// TIA Portal project "Proportional Controller for a Water tank" (V16)
// Vorlageprojekt für das Buch mit Zielsystem S7-1200

(* hardware
DEVICE "S7-1200-Station_1"  S7-1200 Station
   slot 0: "Baugruppenträger_0"  Rack  V1.0
   slot 1: "PLC_1"  CPU 1211C DC/DC/DC  6ES7 211-1AE40-0XB0  V4.1
*)

// ===== PLC "PLC_1"  CPU 1211C DC/DC/DC =====

VAR_GLOBAL   // PLC tag table "Standard-Variablentabelle"
   "xPbStart" AT %I0.0 : Bool;
   "xPbReset" AT %I0.1 : Bool;
   "xPbStop" AT %I0.2 : Bool;
   "xPbStartLed" AT %Q0.0 : Bool;
   "xPbResetLed" AT %Q0.1 : Bool;
   "xPbStopLed" AT %Q0.2 : Bool;
   "rSetpoint" AT %ID38 : Real;
   "rSensorWaterLevel" AT %ID30 : Real;
   "diSP" AT %QD38 : DInt;
   "diPV" AT %QD42 : DInt;
   "rValveFill" AT %QD30 : Real;
   "rValveDischarge" AT %QD34 : Real;
   "xStateStart" AT %M0.0 : Bool;
   "rError" AT %MD2 : Real;
   "rErrorABS" AT %MD6 : Real;
   "rKp" AT %MD10 : Real;
   "rSetpoint_Cm" AT %MD30 : Real;
   "rWaterLevel_Cm" AT %MD34 : Real;
   "xSelectorManual" AT %I0.5 : Bool;
   "xSelectorAuto" AT %I0.4 : Bool;
   "xModeManual" AT %M0.1 : Bool;
   "xModeAuto" AT %M0.2 : Bool;
   "xStep10_EnableRegulator" AT %M0.4 : Bool;
   "xStep30_Discharge" AT %M0.6 : Bool;
   "xStep40_End" AT %M0.7 : Bool;
   "xStep20_LevelCheck" AT %M1.0 : Bool;
   "xAlarm" AT %M0.3 : Bool;
   "xFIOReset" AT %I0.3 : Bool;
   "Clock_Byte" AT %MB100 : Byte;
   "Clock_10Hz" AT %M100.0 : Bool;
   "Clock_5Hz" AT %M100.1 : Bool;
   "Clock_2.5Hz" AT %M100.2 : Bool;
   "Clock_2Hz" AT %M100.3 : Bool;
   "Clock_1.25Hz" AT %M100.4 : Bool;
   "Clock_1Hz" AT %M100.5 : Bool;
   "Clock_0.625Hz" AT %M100.6 : Bool;
   "xPulse" AT %M100.7 : Bool;
   "xStep0_Init" AT %M0.5 : Bool;
   "xMem_0" AT %M1.1 : Bool;
   "diLowerLimit" AT %MD18 : DInt;
   "diupperLimit" AT %MD22 : DInt;
END_VAR

DATA_BLOCK "DB_Regulator"   // DB1
{ S7_Optimized_Access := 'TRUE' }
VERSION : 0.1
   VAR RETAIN
      rKp : Real := 0.1;
   END_VAR
BEGIN
END_DATA_BLOCK

// folder: System blocks/Program resources

DATA_BLOCK "IEC_Timer_0_DB"   // DB2
{ S7_Optimized_Access := 'TRUE' }
AUTHOR : Simatic
FAMILY : IEC
NAME : IEC_TMR
VERSION : 1.0
// stored: InstanceOfName IEC_TIMER
"IEC_TIMER"
BEGIN
END_DATA_BLOCK

// folder: (top level)

FUNCTION "MHJ-PLC-Lab-Function-S71200" : Void   // FC9000, SCL
{ S7_Optimized_Access := 'TRUE' }
VERSION : 0.1
   VAR_TEMP
      rdTimeReturn : Int;
      outputTime : DTL;
      SyncVal : Byte;
      forVal : Int;
      forVal_2 : Int;
      Value : Byte;
   END_VAR
   VAR CONSTANT
      CompVal : Byte := 16#34;
      Value_01 : Byte := 16#11;
      Value_01_DW : DWord := 16#A165_D992;
      Value_02_DW : DWord := 16#58BE_4401;
   END_VAR
BEGIN

   #Value:=PEEK(area := 16#82,
        dbNumber := 0,
        byteOffset := 511);
   #Value := #Value + 1;

   POKE(area := 16#82,
        dbNumber := 0,
        byteOffset := 511,
        value := #Value);

   POKE(area:=16#81,
        dbNumber:=0,
        byteOffset:=1016,
        value:=#Value_01_DW);
   POKE(area := 16#81,
        dbNumber := 0,
        byteOffset := 1020,
        value := #Value_02_DW);

   POKE(area := 16#81,
        dbNumber := 0,
        byteOffset := 511,
        value := B#16#00);

   FOR #forVal := 0 TO 120 DO
       FOR #forVal_2:=0 TO 10 DO
           #rdTimeReturn:=RD_SYS_T(#outputTime);
           #rdTimeReturn := WR_SYS_T(#outputTime);
           #rdTimeReturn := RD_SYS_T(#outputTime);
           #rdTimeReturn := WR_SYS_T(#outputTime);
       END_FOR;
       #SyncVal:= PEEK(area := 16#81,
                      dbNumber := 0,
                      byteOffset := 511);
       IF #SyncVal = #CompVal THEN
          GOTO M_1;
       END_IF;
   END_FOR;
   RETURN;

   M_1:
   POKE(area := 16#81,
        dbNumber := 0,
        byteOffset := 511,
        value := B#16#0);
END_FUNCTION

ORGANIZATION_BLOCK "Main"   // OB1, LAD, ProgramCycle
TITLE = "Main Program Sweep (Cycle)"
{ S7_Optimized_Access := 'TRUE' }
VERSION : 0.1
   VAR_INPUT
      Initial_Call : Bool;   // Initial call of this OB
      Remanence : Bool;   // =True, if remanent data are available
   END_VAR
   VAR_TEMP
      rTemp1 : Real;
      wlevelMeter_2 : Real;
   END_VAR
   VAR_TEMP   // added for the SCL form of the ladder/FBD networks
      _w1 : Bool;
   END_VAR
BEGIN

REGION Network 1: Scaling the set point and current values in CM
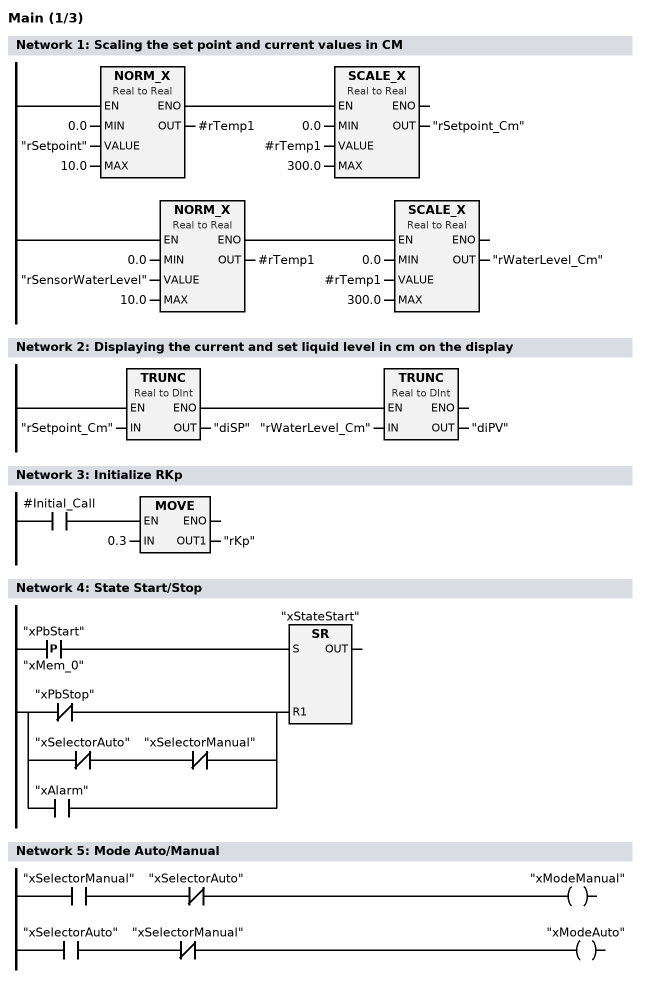
   RUNG wire#powerrail
      { S7_Templates := "[SrcType := Real, DestType := Real]" } Normalize(min := 0.0, value := "rSetpoint", max := 10.0, out => #rTemp1)
      { S7_Templates := "[SrcType := Real, DestType := Real]" } Scale(min := 0.0, value := #rTemp1, max := 300.0, out => "rSetpoint_Cm")
   END_RUNG
   RUNG wire#powerrail
      { S7_Templates := "[SrcType := Real, DestType := Real]" } Normalize(min := 0.0, value := "rSensorWaterLevel", max := 10.0, out => #rTemp1)
      { S7_Templates := "[SrcType := Real, DestType := Real]" } Scale(min := 0.0, value := #rTemp1, max := 300.0, out => "rWaterLevel_Cm")
   END_RUNG
   // the same network as SCL:
   #rTemp1 := NORM_X(MIN := 0.0, VALUE := "rSetpoint", MAX := 10.0);
   "rSetpoint_Cm" := SCALE_X(MIN := 0.0, VALUE := #rTemp1, MAX := 300.0);
   #rTemp1 := NORM_X(MIN := 0.0, VALUE := "rSensorWaterLevel", MAX := 10.0);
   "rWaterLevel_Cm" := SCALE_X(MIN := 0.0, VALUE := #rTemp1, MAX := 300.0);
END_REGION

REGION Network 2: Displaying the current and set liquid level in cm on the display
   RUNG wire#powerrail
      { S7_Templates := "[SrcType := Real, DestType := DInt]" } Trunc(in := "rSetpoint_Cm", out => "diSP")
      { S7_Templates := "[SrcType := Real, DestType := DInt]" } Trunc(in := "rWaterLevel_Cm", out => "diPV")
   END_RUNG
   // the same network as SCL:
   "diSP" := TRUNC("rSetpoint_Cm");
   "diPV" := TRUNC("rWaterLevel_Cm");
END_REGION

REGION Network 3: Initialize RKp
   RUNG wire#powerrail
      Contact( #Initial_Call )
      Move(in := 0.3, out1 => "rKp")
   END_RUNG
   // the same network as SCL:
   IF #Initial_Call THEN "rKp" := 0.3; END_IF;
END_REGION

REGION Network 4: State Start/Stop
   RUNG wire#powerrail
      P_Contact(operand := "xPbStart", bit := "xMem_0")
      S_SR(operand := "xStateStart", r1 := wire#w1)
   END_RUNG
   RUNG wire#powerrail
      I_Contact( "xPbStop" )
   END_RUNG wire#w1
   RUNG wire#powerrail
      I_Contact( "xSelectorAuto" )
      I_Contact( "xSelectorManual" )
   END_RUNG wire#w1
   RUNG wire#powerrail
      Contact( "xAlarm" )
   END_RUNG wire#w1
   // the same network as SCL:
   #_w1 := "xPbStart" AND NOT "xMem_0";   // rising edge of "xPbStart"
   "xMem_0" := "xPbStart";
   IF #_w1 THEN
       "xStateStart" := TRUE;   // SR flip-flop
   END_IF;
   IF NOT "xPbStop" OR (NOT "xSelectorAuto" AND NOT "xSelectorManual") OR "xAlarm" THEN
       "xStateStart" := FALSE;
   END_IF;
END_REGION

REGION Network 5: Mode Auto/Manual
   RUNG wire#powerrail
      Contact( "xSelectorManual" )
      I_Contact( "xSelectorAuto" )
      Coil( "xModeManual" )
   END_RUNG
   RUNG wire#powerrail
      Contact( "xSelectorAuto" )
      I_Contact( "xSelectorManual" )
      Coil( "xModeAuto" )
   END_RUNG
   // the same network as SCL:
   "xModeManual" := "xSelectorManual" AND NOT "xSelectorAuto";
   "xModeAuto" := "xSelectorAuto" AND NOT "xSelectorManual";
END_REGION

REGION Network 6: Scaling the setpoint and current values to a value in cm
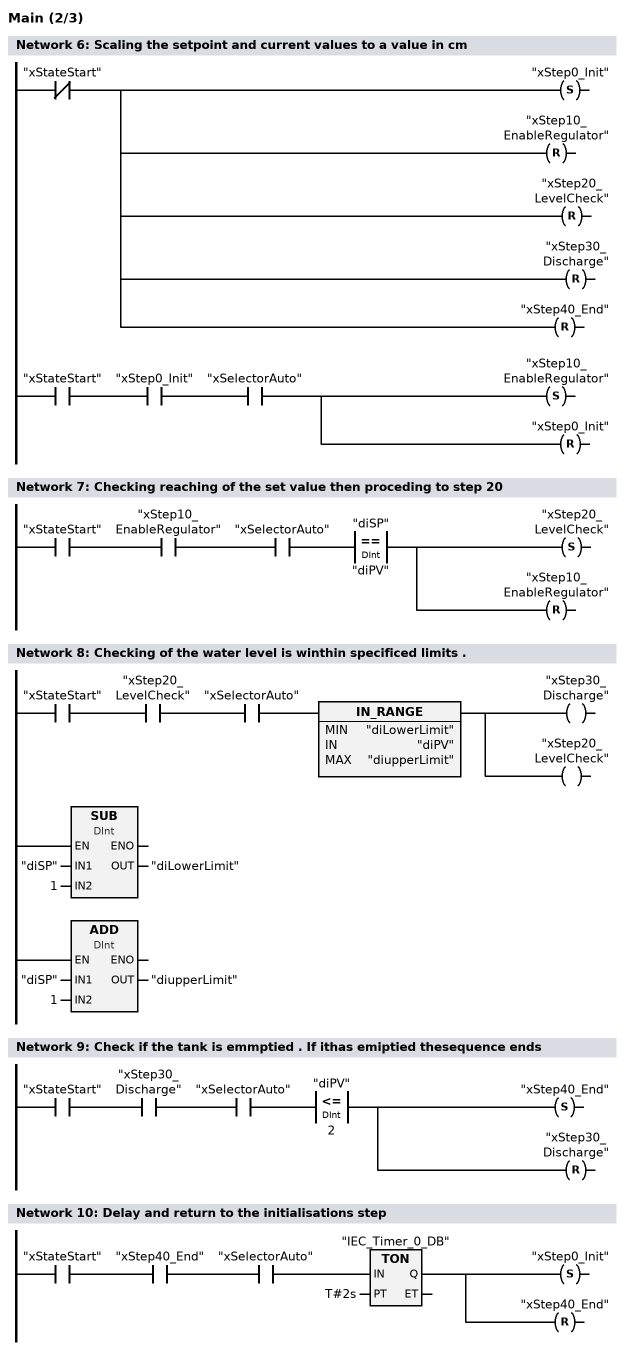
   RUNG wire#powerrail
      I_Contact( "xStateStart" )
      wire#w1
      S_Coil( "xStep0_Init" )
   END_RUNG
   RUNG wire#w1
      R_Coil( "xStep10_EnableRegulator" )
   END_RUNG
   RUNG wire#w1
      R_Coil( "xStep20_LevelCheck" )
   END_RUNG
   RUNG wire#w1
      R_Coil( "xStep30_Discharge" )
   END_RUNG
   RUNG wire#w1
      R_Coil( "xStep40_End" )
   END_RUNG
   RUNG wire#powerrail
      Contact( "xStateStart" )
      Contact( "xStep0_Init" )
      Contact( "xSelectorAuto" )
      wire#w2
      S_Coil( "xStep10_EnableRegulator" )
   END_RUNG
   RUNG wire#w2
      R_Coil( "xStep0_Init" )
   END_RUNG
   // the same network as SCL:
   IF NOT "xStateStart" THEN
       "xStep0_Init" := TRUE;
       "xStep10_EnableRegulator" := FALSE;
       "xStep20_LevelCheck" := FALSE;
       "xStep30_Discharge" := FALSE;
       "xStep40_End" := FALSE;
   END_IF;
   IF "xStateStart" AND "xStep0_Init" AND "xSelectorAuto" THEN
       "xStep10_EnableRegulator" := TRUE;
       "xStep0_Init" := FALSE;
   END_IF;
END_REGION

REGION Network 7: Checking reaching of the set value then proceding to step 20
   RUNG wire#powerrail
      Contact( "xStateStart" )
      Contact( "xStep10_EnableRegulator" )
      Contact( "xSelectorAuto" )
      { S7_Templates := "SrcType := DInt" } EQ_Contact(in1 := "diSP", in2 := "diPV")
      wire#w1
      S_Coil( "xStep20_LevelCheck" )
   END_RUNG
   RUNG wire#w1
      R_Coil( "xStep10_EnableRegulator" )
   END_RUNG
   // the same network as SCL:
   IF "xStateStart" AND "xStep10_EnableRegulator" AND "xSelectorAuto" AND ("diSP" = "diPV") THEN
       "xStep20_LevelCheck" := TRUE;
       "xStep10_EnableRegulator" := FALSE;
   END_IF;
END_REGION

REGION Network 8: Checking of the water level is winthin specificed limits .
   RUNG wire#powerrail
      Contact( "xStateStart" )
      Contact( "xStep20_LevelCheck" )
      Contact( "xSelectorAuto" )
      { S7_Templates := "SrcType := DInt" } InRange(min := "diLowerLimit", in := "diPV", max := "diupperLimit")
      wire#w1
      Coil( "xStep30_Discharge" )
   END_RUNG
   RUNG wire#w1
      Coil( "xStep20_LevelCheck" )
   END_RUNG
   RUNG wire#powerrail
      { S7_Templates := "SrcType := DInt" } Sub(in1 := "diSP", in2 := 1, out => "diLowerLimit")
   END_RUNG
   RUNG wire#powerrail
      { S7_Templates := "SrcType := DInt" } Add(in1 := "diSP", in2 := 1, out => "diupperLimit")
   END_RUNG
   // the same network as SCL:
   "xStep30_Discharge" := "xStateStart" AND "xStep20_LevelCheck" AND "xSelectorAuto" AND ("diLowerLimit" <= "diPV") AND ("diPV" <= "diupperLimit");
   "xStep20_LevelCheck" := "xStep30_Discharge";
   "diLowerLimit" := "diSP" - 1;
   "diupperLimit" := "diSP" + 1;
END_REGION

REGION Network 9: Check if the tank is emmptied . If ithas emiptied thesequence ends
   RUNG wire#powerrail
      Contact( "xStateStart" )
      Contact( "xStep30_Discharge" )
      Contact( "xSelectorAuto" )
      { S7_Templates := "SrcType := DInt" } LE_Contact(in1 := "diPV", in2 := 2)
      wire#w1
      S_Coil( "xStep40_End" )
   END_RUNG
   RUNG wire#w1
      R_Coil( "xStep30_Discharge" )
   END_RUNG
   // the same network as SCL:
   IF "xStateStart" AND "xStep30_Discharge" AND "xSelectorAuto" AND ("diPV" <= 2) THEN
       "xStep40_End" := TRUE;
       "xStep30_Discharge" := FALSE;
   END_IF;
END_REGION

REGION Network 10: Delay and return to the initialisations step
   "IEC_Timer_0_DB".TON(IN := "xStateStart" AND "xStep40_End" AND "xSelectorAuto", PT := T#2s);
   IF "IEC_Timer_0_DB".Q THEN
       "xStep0_Init" := TRUE;
       "xStep40_End" := FALSE;
   END_IF;
END_REGION

REGION Network 11: Alarm and stop the sequence auto
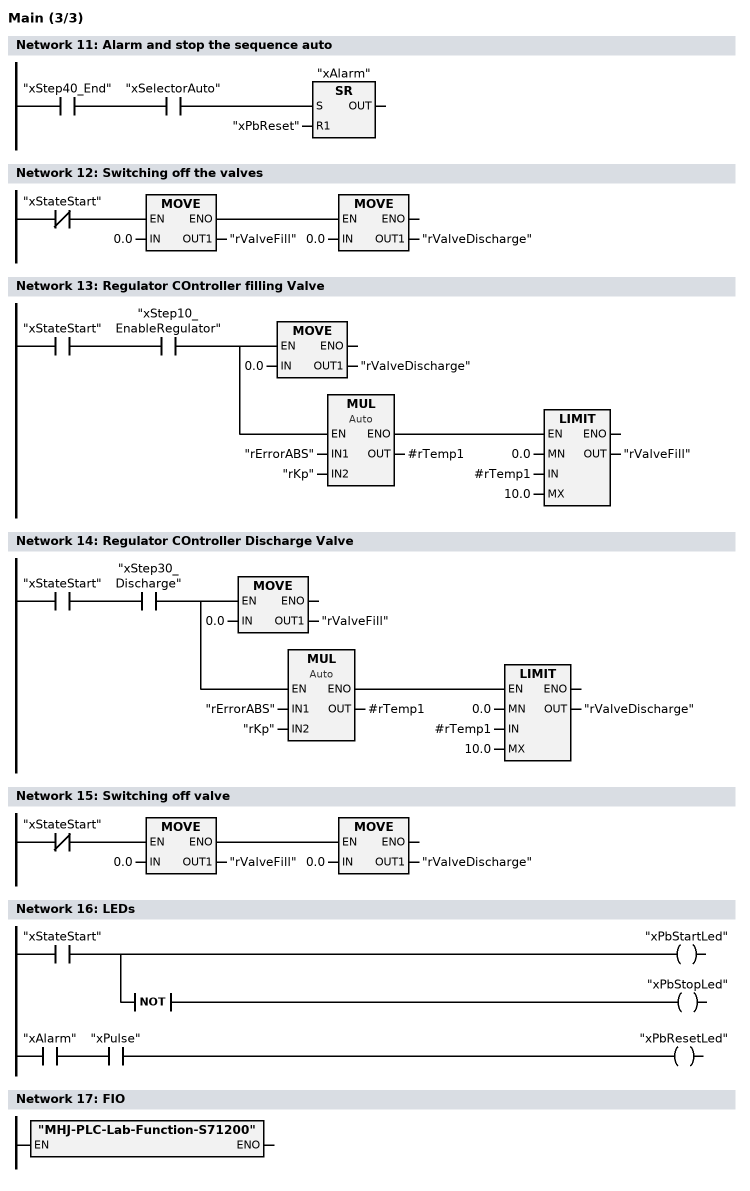
   RUNG wire#powerrail
      Contact( "xStep40_End" )
      Contact( "xSelectorAuto" )
      S_SR(operand := "xAlarm", r1 := "xPbReset")
   END_RUNG
   // the same network as SCL:
   IF "xStep40_End" AND "xSelectorAuto" THEN
       "xAlarm" := TRUE;   // SR flip-flop
   END_IF;
   IF "xPbReset" THEN "xAlarm" := FALSE; END_IF;
END_REGION

REGION Network 12: Switching off the valves
   RUNG wire#powerrail
      I_Contact( "xStateStart" )
      Move(in := 0.0, out1 => "rValveFill")
      Move(in := 0.0, out1 => "rValveDischarge")
   END_RUNG
   // the same network as SCL:
   IF NOT "xStateStart" THEN
       "rValveFill" := 0.0;
       "rValveDischarge" := 0.0;
   END_IF;
END_REGION

REGION Network 13: Regulator COntroller filling Valve
   IF "xStateStart" AND "xStep10_EnableRegulator" THEN
       "rValveDischarge" := 0.0;
       #rTemp1 := "rErrorABS" * "rKp";
       "rValveFill" := LIMIT(MN := 0.0, IN := #rTemp1, MX := 10.0);
   END_IF;
END_REGION

REGION Network 14: Regulator COntroller Discharge Valve
   IF "xStateStart" AND "xStep30_Discharge" THEN
       "rValveFill" := 0.0;
       #rTemp1 := "rErrorABS" * "rKp";
       "rValveDischarge" := LIMIT(MN := 0.0, IN := #rTemp1, MX := 10.0);
   END_IF;
END_REGION

REGION Network 15: Switching off valve
   RUNG wire#powerrail
      I_Contact( "xStateStart" )
      Move(in := 0.0, out1 => "rValveFill")
      Move(in := 0.0, out1 => "rValveDischarge")
   END_RUNG
   // the same network as SCL:
   IF NOT "xStateStart" THEN
       "rValveFill" := 0.0;
       "rValveDischarge" := 0.0;
   END_IF;
END_REGION

REGION Network 16: LEDs
   RUNG wire#powerrail
      Contact( "xStateStart" )
      wire#w1
      Coil( "xPbStartLed" )
   END_RUNG
   RUNG wire#w1
      Not()
      Coil( "xPbStopLed" )
   END_RUNG
   RUNG wire#powerrail
      Contact( "xAlarm" )
      Contact( "xPulse" )
      Coil( "xPbResetLed" )
   END_RUNG
   // the same network as SCL:
   "xPbStartLed" := "xStateStart";
   "xPbStopLed" := NOT "xStateStart";
   "xPbResetLed" := "xAlarm" AND "xPulse";
END_REGION

REGION Network 17: FIO
   RUNG wire#powerrail
      "MHJ-PLC-Lab-Function-S71200"()
   END_RUNG
   // the same network as SCL:
   "MHJ-PLC-Lab-Function-S71200"();
END_REGION
END_ORGANIZATION_BLOCK